Universal Robots PolyScope program: tvt19spl_auton_tunnistus_3.urp

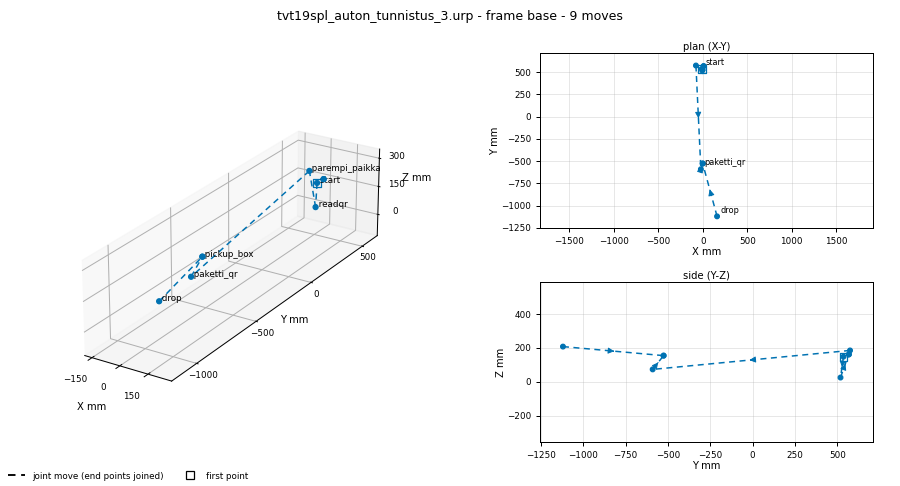
[picture p0: tool path of tvt19spl_auton_tunnistus_3.urp in frame base, 9 of 13 moves have a stored position in this frame; points joined in program order, loops and branches not executed]
Program tvt19spl_auton_tunnistus_3 (installation=default directory=/programs/usbdisk_1/TVT19SPL createdIn=5.11.5.1010327 lastSavedIn=5.11.5.1010327 robotSerialNumber=20195600355)
Calibrated DH parameters: a=[0.000056, -0.161146, -0.252643, 0.000052, -0.000071, 0]; d=[0.181245, -342.672485, 975.135632, -632.288651, 0.119957, 0.115765]; alpha=[1.571164, 0.001314, -0.000405, 1.570615, -1.570559, 0]; deltaTheta=[0, -1.227166, 0.434415, 0.792759, -0.000001, 0]
Robot Program (runOnlyOnce=false)
